// TwinCAT 3 PLC project PLC1
// ProgramVersion: 3.1.4023.0
// libraries:
//   Tc2_Math, * (Beckhoff Automation GmbH)
//   Tc2_Standard, * (Beckhoff Automation GmbH)
//   Tc2_System, * (Beckhoff Automation GmbH)
//   Tc2_Utilities, * (Beckhoff Automation GmbH)
//   Tc3_Module, * (Beckhoff Automation GmbH)
// project tree:
//   Checks/ CheckBounds.TcPOU, CheckDivDInt.TcPOU, CheckDivLInt.TcPOU, CheckDivLReal.TcPOU, CheckDivReal.TcPOU, CheckLRangeSigned.TcPOU, CheckLRangeUnsigned.TcPOU, CheckPointer.TcPOU, CheckRangeSigned.TcPOU, CheckRangeUnsigned.TcPOU
//   FBs/ FB_Env.TcPOU, FB_QAgent.TcPOU
//   / PlcTask.TcTTO
//   POUs/ MAIN.TcPOU
//   STM/ E_STM_QLearning.TcDUT, E_STM_STEP.TcDUT
// real-time tasks:
//   TASK PlcTask: cycle T#2ms, priority 20, ADS port 350

CONFIGURATION PLC1
    RESOURCE PLC ON TwinCAT3
        TASK PlcTask(INTERVAL := T#2ms, PRIORITY := 20);
        PROGRAM MAIN WITH PlcTask : MAIN;
    END_RESOURCE
END_CONFIGURATION

// ---- STM/E_STM_QLearning.TcDUT
{attribute 'qualified_only'}
{attribute 'strict'}
TYPE E_STM_QLearning :
(
	init := 0,
	reset,
	resetWaitOK,
	step,
	stepOK,
	compute,
	computeOK,
	playEnvironment,
	donePlayingEnvironment
);
END_TYPE

// ---- STM/E_STM_STEP.TcDUT
{attribute 'qualified_only'}
{attribute 'strict'}
TYPE E_STM_STEP :
(
	resetEnv := 0,
	computeAction,
	executeAction,
	updateQtable,
	trackReward,
	updateState,
	checkIfDone
);
END_TYPE

// ---- POUs/MAIN.TcPOU
PROGRAM MAIN
VAR
	eSTM_QLearning : E_STM_QLearning;
	eSTM_STEP : E_STM_STEP ;
	FB_QAgent1 : FB_QAgent; // The Q agent will try to solve the Cliffwalking environment
	FB_Env1 : FB_Env := (sPathToBatchFile := 'C:\Users\BramS\Downloads\GitHubPrjs\ST_QLearning\Python\batch.bat',
						sPathToBatchFileFolder := 'C:\Users\BramS\Downloads\GitHubPrjs\ST_QLearning\Python');
	actualEpisode: INT;
	actualStep : INT;
	state : INT;
	actionToTake : INT;
	newState: INT;
	reward: INT;
	done : BOOL;
	aRewardsPerEpisode : ARRAY[0..1000] OF INT;
END_VAR

CASE eSTM_QLearning OF 
     E_STM_QLearning.init:
		FB_QAgent1.M_Init(Alpha := 0.9, Gamma := 0.8, Epsilon := 0.9999, Decay := 0.999);
		FB_Env1.M_StartProxy();
		IF FB_Env1.bStartProxyOK THEN
			eSTM_QLearning := E_STM_QLearning.playEnvironment;
		END_IF
     E_STM_QLearning.playEnvironment :
		IF actualEpisode < 1000 THEN
			IF actualStep <200 THEN
				CASE eSTM_STEP OF
					E_STM_STEP.resetEnv:
						FB_Env1.M_ResetEnvironment();
						IF FB_Env1.bResetEnvironmentOK THEN
							FB_Env1.M_ConfirmEnvResetRead();
							state := FB_Env1.state;
							eSTM_STEP := E_STM_STEP.computeAction;
						END_IF
					E_STM_STEP.computeAction:
						// Update step counter
						actualStep := actualStep + 1;
						actionToTake := FB_QAgent1.M_ComputeAction(state);
						eSTM_STEP := E_STM_STEP.executeAction;
					E_STM_STEP.executeAction:
						FB_Env1.M_Step(actionToTake);
						IF FB_Env1.bEnvStepRequestedOK THEN
							FB_Env1.M_ConfirmEnvStepRequestRead();
							newState := FB_Env1.newState;
							reward := FB_Env1.reward;
							done := FB_Env1.done;
							eSTM_STEP := E_STM_STEP.updateQtable;
						END_IF			
					E_STM_STEP.updateQtable:
						// improved reward function
						IF newState = state THEN
							reward := -100;
						END_IF
						FB_QAgent1.M_ComputeQTable(actionToTake, reward, state, newState);
						eSTM_STEP := E_STM_STEP.trackReward;
					E_STM_STEP.trackReward:
						aRewardsPerEpisode[actualEpisode] := aRewardsPerEpisode[actualEpisode]+reward;
						eSTM_STEP := E_STM_STEP.updateState;
					E_STM_STEP.updateState:
						state := newState;
						eSTM_STEP := E_STM_STEP.checkIfDone;
					E_STM_STEP.checkIfDone:
						IF done THEN
							// The agent has reached the target
							done := FALSE;
							eSTM_STEP := E_STM_STEP.resetEnv;
							FB_Env1.M_ResetInternalStates();
							actualStep := 0;
							actualEpisode := actualEpisode +1;
						ELSE
							eSTM_STEP := E_STM_STEP.computeAction;							
						END_IF
				END_CASE
			ELSE
				// The agent has taken more than 200 steps
				eSTM_STEP := E_STM_STEP.resetEnv;
				FB_Env1.M_ResetInternalStates();
				actualStep := 0;
				actualEpisode := actualEpisode +1;				
			END_IF
		ELSE
			// more than 1000 episodes have passed
			FB_Env1.M_StopEnvironment();
			actualStep := 0;
			
		END_IF
	ELSE 
		eSTM_QLearning := E_STM_QLearning.donePlayingEnvironment;
END_CASE;

FB_Env1();
FB_QAgent1();

END_PROGRAM

// ---- FBs/FB_QAgent.TcPOU
FUNCTION_BLOCK FB_QAgent
VAR_INPUT

END_VAR
VAR_OUTPUT

END_VAR
VAR CONSTANT
	nr_states 	: INT 		:= 48;
	nr_actions 	: INT 		:= 4;	
END_VAR
VAR
	_alpha 		: LREAL 	:= 0.2;
	_gamma 		: LREAL 	:= 0.5;
	_epsilon 	: LREAL 	:= 1;
	_decay 		: LREAL 	:= 0.99;
	_r			: LREAL     := 0;
	_actionToTake : INT;
	_state 		: INT :=  0;
	_reward 	: INT;
	_newState	: INT;
	_possibleActions : ARRAY[0..nr_actions-1] OF INT := [0,1,2,3];
	_q_table : ARRAY[0..nr_states-1] OF ARRAY[0..nr_actions-1] OF REAL;
	DRAND : DRAND;
END_VAR
VAR_IN_OUT

END_VAR

METHOD PUBLIC M_ComputeAction : INT
VAR_INPUT
	State : INT;
END_VAR
VAR
	tempRandomValue : LREAL;
	tempCounter : INT;
	tempHighestIndex : INT;
END_VAR
_epsilon := _epsilon*_decay;
DRAND(Seed:= 2, Num=> _r);
IF _r <= _epsilon THEN
	// EXPLORE: Find random action
	DRAND(Seed:= 2, Num=> tempRandomValue);
	tempRandomValue := tempRandomValue*nr_actions;
	tempRandomValue := FLOOR(tempRandomValue);
	M_ComputeAction := 	_possibleActions[TO_INT(tempRandomValue)];
	

ELSE
	// EXPLOIT: Find action with highest Q Value
	tempHighestIndex := 0;
	FOR tempCounter:=0 TO (nr_actions-1) BY 1 DO
    	IF _q_table[State][tempCounter] >_q_table[State][tempHighestIndex] THEN
			tempHighestIndex := tempCounter;
		END_IF
	END_FOR;
	M_ComputeAction := tempHighestIndex;	
END_IF
END_METHOD

METHOD PUBLIC M_ComputeQTable 
VAR_INPUT
	actionToTake : INT;
	reward 	: INT;
	state 		: INT;
	newState 	: INT;
END_VAR
VAR
	tempHighestIndex : INT;
	tempCounter : INT;
	oldReward, newReward,discountFutureReward: REAL;
END_VAR
_reward := reward;
_state := state; 
_newState := newState;
_actionToTake := actionToTake;
									
// Find future action with highest value in newState
tempHighestIndex := 0;
FOR tempCounter:=0 TO (nr_actions-1) BY 1 DO
	IF _q_table[newState][tempCounter] >_q_table[newState][tempHighestIndex] THEN
		tempHighestIndex := tempCounter;
	END_IF
END_FOR;

// Waarde van de gekozen actie in de huidige state bijwerken
_q_table[_state][_actionToTake] := TO_REAL((1-_alpha)*_q_table[_state][_actionToTake] + _alpha*(_reward+_gamma*(_q_table[_newState][tempHighestIndex])));
END_METHOD

METHOD PUBLIC M_Init : BOOL
VAR_INPUT
	Alpha 	: LREAL;
	Gamma 	: LREAL;
	Epsilon : LREAL;
	Decay 	: LREAL;
END_VAR
_alpha 		:= Alpha;
_gamma 		:= Gamma;
_epsilon 	:= Epsilon;
_decay 		:= Decay;
END_METHOD

METHOD M_SaveWeights
VAR_INPUT
END_VAR
// TODO: Export to JSON
END_METHOD

END_FUNCTION_BLOCK

// ---- FBs/FB_Env.TcPOU
FUNCTION_BLOCK FB_Env
(*
	The environment should provide methods like step, reset etc...
	If the environment is outside of the PLC environment, it should act like a proxy, or contact one
*)
VAR_INPUT
END_VAR
VAR_OUTPUT
	bResetEnvironmentOK : BOOL;
	bStartProxyOK : BOOL;
	bEnvStepRequestedOK : BOOL;
	state : INT;
	newState : INT;
	reward : INT;
	done : BOOL;
END_VAR
VAR
	_bEnvResetRequested : BOOL;
	_bProxyStarted : BOOL;
	_bEnvStepRequested : BOOL;
	_bStopEnvironmentRequested : BOOL;
	_actionToTake : INT;
	startProxy : NT_StartProcess;
	sPathToBatchFile : STRING;
	sPathToBatchFileFolder : STRING;
END_VAR

startProxy(
	NETID:= '', 
	PATHSTR:= sPathToBatchFile, 
	DIRNAME:= sPathToBatchFileFolder, 
	COMNDLINE:= , 
	START:= FALSE, 
	TMOUT:= , 
	BUSY=> , 
	ERR=> , 
	ERRID=> );

METHOD M_ConfirmEnvResetRead
VAR_INPUT
END_VAR
bResetEnvironmentOK := FALSE;
_bEnvResetRequested := FALSE;
END_METHOD

METHOD M_ConfirmEnvStepRequestRead
VAR_INPUT
END_VAR
bEnvStepRequestedOK := FALSE;
_bEnvStepRequested := FALSE;
END_METHOD

METHOD PUBLIC M_ResetEnvironment
VAR_INPUT
END_VAR
IF NOT _bEnvResetRequested THEN
	_bEnvResetRequested := TRUE;
END_IF
END_METHOD

METHOD M_ResetInternalStates
VAR_INPUT
END_VAR
bResetEnvironmentOK := FALSE;
bStartProxyOK := FALSE;
bEnvStepRequestedOK := FALSE;
done := FALSE;
_bEnvResetRequested := FALSE;
_bEnvStepRequested := FALSE;
END_METHOD

METHOD PUBLIC M_StartProxy : BOOL
VAR_INPUT
END_VAR
IF NOT _bProxyStarted THEN
	_bProxyStarted := TRUE;
	startProxy(
		NETID:= '', 
		PATHSTR:= sPathToBatchFile, 
		DIRNAME:= sPathToBatchFileFolder, 
		COMNDLINE:= , 
		START:= TRUE, 
		TMOUT:= , 
		BUSY=> , 
		ERR=> , 
		ERRID=> );
END_IF
END_METHOD

METHOD M_Step 
VAR_INPUT
	actionToTake : INT;
END_VAR
IF NOT _bEnvStepRequested THEN
	_actionToTake := actionToTake;
	_bEnvStepRequested := TRUE;
END_IF
END_METHOD

METHOD M_StopEnvironment
VAR_INPUT
END_VAR
IF NOT _bStopEnvironmentRequested THEN
	_bStopEnvironmentRequested := TRUE;
END_IF
END_METHOD

END_FUNCTION_BLOCK

// ---- Checks/CheckBounds.TcPOU
// Implicitly generated code : DO NOT EDIT
FUNCTION CheckBounds : DINT
VAR_INPUT
	index, lower, upper: DINT;
END_VAR

// Implicitly generated code : Only an Implementation suggestion
{noflow}
IF  index < lower THEN
	CheckBounds := lower;
ELSIF  index > upper THEN
	CheckBounds := upper;
ELSE  
	CheckBounds := index;
END_IF
{flow}

END_FUNCTION

// ---- Checks/CheckDivDInt.TcPOU
// Implicitly generated code : DO NOT EDIT
FUNCTION CheckDivDInt : DINT
VAR_INPUT
	divisor:DINT;
END_VAR

// Implicitly generated code : Only an Implementation suggestion
{noflow}
IF divisor = 0 THEN
	CheckDivDInt:=1;
ELSE
	CheckDivDInt:=divisor;
END_IF;
{flow}

END_FUNCTION

// ---- Checks/CheckDivLInt.TcPOU
// Implicitly generated code : DO NOT EDIT
FUNCTION CheckDivLInt : LINT
VAR_INPUT
	divisor:LINT;
END_VAR

// Implicitly generated code : Only an Implementation suggestion
{noflow}
IF divisor = 0 THEN
	CheckDivLInt:=1;
ELSE
	CheckDivLInt:=divisor;
END_IF;
{flow}

END_FUNCTION

// ---- Checks/CheckDivLReal.TcPOU
// Implicitly generated code : DO NOT EDIT
FUNCTION CheckDivLReal : LREAL
VAR_INPUT
	divisor:LREAL;
END_VAR

// Implicitly generated code : Only an Implementation suggestion
{noflow}
IF divisor = 0 THEN
	CheckDivLReal:=1;
ELSE
	CheckDivLReal:=divisor;
END_IF;
{flow}

END_FUNCTION

// ---- Checks/CheckDivReal.TcPOU
// Implicitly generated code : DO NOT EDIT
FUNCTION CheckDivReal : REAL
VAR_INPUT
	divisor:REAL;
END_VAR

// Implicitly generated code : Only an Implementation suggestion
{noflow}
IF divisor = 0 THEN
	CheckDivReal:=1;
ELSE
	CheckDivReal:=divisor;
END_IF;
{flow}

END_FUNCTION

// ---- Checks/CheckLRangeSigned.TcPOU
// Implicitly generated code : DO NOT EDIT
FUNCTION CheckLRangeSigned : LINT
VAR_INPUT
	value, lower, upper: LINT;
END_VAR

// Implicitly generated code : Only an Implementation suggestion
{noflow}
IF (value < lower) THEN
	CheckLRangeSigned := lower;
ELSIF(value > upper) THEN
	CheckLRangeSigned := upper;
ELSE
	CheckLRangeSigned := value;
END_IF

{flow}

END_FUNCTION

// ---- Checks/CheckLRangeUnsigned.TcPOU
// Implicitly generated code : DO NOT EDIT
FUNCTION CheckLRangeUnsigned : ULINT
VAR_INPUT
	value, lower, upper: ULINT;
END_VAR

// Implicitly generated code : Only an Implementation suggestion
{noflow}
IF (value < lower) THEN
	CheckLRangeUnsigned := lower;
ELSIF(value > upper) THEN
	CheckLRangeUnsigned := upper;
ELSE
	CheckLRangeUnsigned := value;
END_IF
{flow}

END_FUNCTION

// ---- Checks/CheckPointer.TcPOU
// Implicitly generated code : DO NOT EDIT
FUNCTION CheckPointer : POINTER TO BYTE
VAR_INPUT 
	ptToTest : POINTER TO BYTE; // Destination address of the pointer
	iSize : DINT;		        // Size of the type the pointer points to. (e.g: 20 for POINTER TO ARRAY [0..9] OF INT) 
	iGran : DINT;		        // Granularity of the pointer access. This is the size of the biggest non-structured data type in the type the pointer points to. (e.g: 2 for POINTER TO ARRAY [0..9] OF INT)
	bWrite: BOOL;		        // Indicates read or write Access. TRUE = write access.
END_VAR

// Implicitly generated code : Only an Implementation suggestion
{noflow}
IF ptToTest=0 THEN
    ADSLOGSTR(ADSLOG_MSGTYPE_ERROR OR ADSLOG_MSGTYPE_STRING,'CheckPointer failed due to invalid address.','');
ELSIF iSize<=0 THEN
    ADSLOGSTR(ADSLOG_MSGTYPE_ERROR OR ADSLOG_MSGTYPE_STRING,'CheckPointer failed due to invalid size.','');
ELSIF iGran<=0 THEN
    ADSLOGSTR(ADSLOG_MSGTYPE_ERROR OR ADSLOG_MSGTYPE_STRING,'CheckPointer failed due to invalid granularity.','');
// -> Please note that the following memory area check is time consuming:
//ELSIF F_CheckMemoryArea(pData:=ptToTest,nSize:=DINT_TO_UDINT(iSize)) = E_TcMemoryArea.Unknown THEN
//    ADSLOGSTR(ADSLOG_MSGTYPE_ERROR OR ADSLOG_MSGTYPE_STRING,'CheckPointer failed due to unknown memory area.','');
END_IF
CheckPointer := ptToTest;
{flow}

END_FUNCTION

// ---- Checks/CheckRangeSigned.TcPOU
// Implicitly generated code : DO NOT EDIT
FUNCTION CheckRangeSigned : DINT
VAR_INPUT
	value, lower, upper: DINT;
END_VAR

// Implicitly generated code : Only an Implementation suggestion
{noflow}
IF (value < lower) THEN
	CheckRangeSigned := lower;
ELSIF(value > upper) THEN
	CheckRangeSigned := upper;
ELSE
	CheckRangeSigned := value;
END_IF
{flow}

END_FUNCTION

// ---- Checks/CheckRangeUnsigned.TcPOU
// Implicitly generated code : DO NOT EDIT
FUNCTION CheckRangeUnsigned : UDINT
VAR_INPUT
	value, lower, upper: UDINT;
END_VAR

// Implicitly generated code : Only an Implementation suggestion
{noflow}
IF (value < lower) THEN
	CheckRangeUnsigned := lower;
ELSIF(value > upper) THEN
	CheckRangeUnsigned := upper;
ELSE
	CheckRangeUnsigned := value;
END_IF
{flow}

END_FUNCTION
